FUNCTION_BLOCK ARRAY2ARRAY_8_INT (* Service Interface Function Block Type *)
  (* Description: Copyright (c) 2014 Profactor GmbH, HR Agrartechnik GmbH This program and the accompanying materials are made available under the terms of the Eclipse Public License 2.0 which is available at https://www.eclipse.org/legal/epl-2.0/ SPDX-License-Identifier: EPL-2.0 *)
  (* Version 1.0, 2026-03-30, Franz Höpfinger, HR Agrartechnik GmbH, copy ARRAY2ARRAY_2_LREAL and made this block *)
  PACKAGE eclipse4diac::convert;
  {SET_ATTRIBUTE(eclipse4diac::core::GenericClassName, 'GEN_ARRAY2ARRAY')}
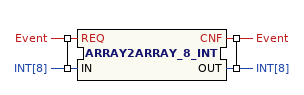
  EVENT_INPUT
    REQ WITH IN; (* Service Request *)
  END_EVENT
  EVENT_OUTPUT
    CNF WITH OUT; (* Confirmation of Requested Service *)
  END_EVENT
  VAR_INPUT
    IN : ARRAY [0..7] OF INT; (* array input *)
  END_VAR
  VAR_OUTPUT
    OUT : ARRAY [0..7] OF INT; (* array output *)
  END_VAR
END_FUNCTION_BLOCK
